// TwinCAT 3 PLC project Itsanewproject
// ProgramVersion: 3.1.4024.0
// libraries:
//   Tc2_Standard, * (Beckhoff Automation GmbH)
//   Tc2_System, * (Beckhoff Automation GmbH)
//   Tc3_Module, * (Beckhoff Automation GmbH)
// project tree:
//   / PlcTask.TcTTO
//   POUs/ Lamp.TcPOU, Light.TcPOU, MAIN.TcPOU
// real-time tasks:
//   TASK PlcTask: cycle T#10ms, priority 20, ADS port 350
// I/O:
//   DEVICE Device 1 (EtherCAT), AmsNetId 10.200.224.204.2.1
//     Term 1 (EK1100) [EK1100 EtherCAT Coupler (2A E-Bus)]

CONFIGURATION Itsanewproject
    RESOURCE PLC ON TwinCAT3
        TASK PlcTask(INTERVAL := T#10ms, PRIORITY := 20);
        PROGRAM MAIN WITH PlcTask : MAIN;
    END_RESOURCE
END_CONFIGURATION

// ---- POUs/MAIN.TcPOU
PROGRAM MAIN
VAR
	input :BOOL;
	output : BOOL;
	
END_VAR

Lamp ();
Light();

END_PROGRAM

// ---- POUs/Lamp.TcPOU
PROGRAM Lamp
VAR
	counter11 : int;
END_VAR

counter11 := counter11 + 1;

END_PROGRAM

// ---- POUs/Light.TcPOU
PROGRAM Light
VAR
	counter : int;
END_VAR

counter := counter + 11;

END_PROGRAM
